PROGRAM MAIN
VAR
	Festo : Festo_IoLink_VacumEjector_OVEM_H_CE;
	Execute: BOOL;
	amsNetId : AMSNETID;
	netid : T_AmsNetIdAr;
END_VAR

ACTION IO_Link:
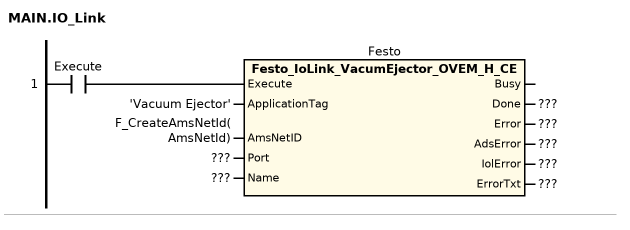
// NETWORK 1
Festo(Execute := Execute, ApplicationTag := 'Vacuum Ejector', AmsNetID := F_CreateAmsNetId(AmsNetId)); // Festo_IoLink_VacumEjector_OVEM_H_CE
END_ACTION

END_PROGRAM

(* stored: Version 1.1.0.1, ProductVersion 3.1.4024.11
   POU MAIN: Id {c0a69bbd-f10e-4371-b8f4-dcd0f6bb0d31}, SpecialFunc None
   Action IO_Link: Id {849431fe-ca07-4d14-a60e-5c9c0c19d635} *)
